FUNCTION_BLOCK FB_XtsXlMoverUtility
VAR_INPUT
	EdtDriverOid: OTCID;
END_VAR

VAR_OUTPUT
	bBusy: BOOL;
	bDone: BOOL;
	bError: BOOL;
	bInit: BOOL;
	ipResultMessage: I_TcMessage := fbResult;
END_VAR

VAR
	fbResult: FB_TcMessage;
	_ipComObject: ITComObject;
	
	PID_TriggerLeave						: PTCID := 16#030802EF;
	PID_TriggerArrive						: PTCID := 16#030802EE;
	PID_IsVirtualFeedbackEnabled			: PTCID := 16#0308050B;
	PID_ConfiguredDetectionTrackObjectId	: PTCID := 16#030802F0;
	PID_StartupTrackPosition				: PTCID := 16#03080370;
END_VAR

IF NOT bInit THEN
	IF GetComObject(nObjectId:=EdtDriverOid) THEN
		bInit:=TRUE;
	END_IF
	RETURN;
END_IF

METHOD GetComObject : BOOL
VAR_INPUT
	nObjectId: OTCID;
END_VAR
IF FW_ObjMgr_GetObjectInstance(	oid		:= nObjectId, 
								iid		:= TC_GLOBAL_IID_LIST.IID_ITComObject, 
								pipUnk	:= ADR(_ipComObject)) = 0
THEN
	GetComObject := TRUE;
END_IF
END_METHOD

METHOD SetConfiguredDetectionTrackObjectId : BOOL
VAR_INPUT
	nConfiguredDetectionTrackObjectId: OTCID;
END_VAR

VAR
	nValue: OTCID;
	stEventEntry: TcEventEntry;
	pstEventEntry: REFERENCE TO TcEventEntry := stEventEntry;
END_VAR

VAR_INST
	hResult : HRESULT;
END_VAR
bError := FALSE;

nValue := nConfiguredDetectionTrackObjectId;

IF _ipComObject <> 0 THEN 
	 hResult := 	_ipComObject.TcSetObjPara(		pid := PID_ConfiguredDetectionTrackObjectId,
													nData := SIZEOF(nValue),
													pData := ADR(nValue),
													pgp := 0); 	
	IF hResult = 0 THEN
		SetConfiguredDetectionTrackObjectId := TRUE;
	ELSE
		HRESULTAdsErr_TO_TcEventEntry(hResult,stEventEntry);
		IF NOT fbResult.EqualsToEventEntryEx( stOther := stEventEntry) THEN
			fbResult.CreateEx(stEventEntry, 0);
			fbResult.Send(0);
			fbResult.Release();
		END_IF
		bError := TRUE;
	END_IF							
END_IF
END_METHOD

METHOD SetIsVirtualFeedbackEnabled : BOOL
VAR_INPUT
	bSetIsVirtualFeedbackEnabled: BOOL;
END_VAR

VAR
	nValue: BOOL;
	stEventEntry: TcEventEntry;
	pstEventEntry: REFERENCE TO TcEventEntry := stEventEntry;
END_VAR

VAR_INST
	hResult : HRESULT;
END_VAR
bError := FALSE;

nValue := bSetIsVirtualFeedbackEnabled;

IF _ipComObject <> 0 THEN 
	 hResult := 	_ipComObject.TcSetObjPara(		pid := PID_IsVirtualFeedbackEnabled,
													nData := SIZEOF(nValue),
													pData := ADR(nValue),
													pgp := 0); 	
	IF hResult = 0 THEN
		SetIsVirtualFeedbackEnabled := TRUE;
	ELSE
		HRESULTAdsErr_TO_TcEventEntry(hResult,stEventEntry);
		IF NOT fbResult.EqualsToEventEntryEx( stOther := stEventEntry) THEN
			fbResult.CreateEx(stEventEntry, 0);
			fbResult.Send(0);
			fbResult.Release();
		END_IF
		bError := TRUE;
	END_IF							
END_IF
END_METHOD

METHOD SetStartupTrackPosition : BOOL
VAR_INPUT
	nStartupTrackPosition: REAL;
END_VAR

VAR
	nValue: REAL;
	stEventEntry: TcEventEntry;
	pstEventEntry: REFERENCE TO TcEventEntry := stEventEntry;
END_VAR

VAR_INST
	hResult : HRESULT;
END_VAR
bError := FALSE;

nValue := nStartupTrackPosition;

IF _ipComObject <> 0 THEN 
	 hResult := 	_ipComObject.TcSetObjPara(		pid := PID_StartupTrackPosition,
													nData := SIZEOF(nValue),
													pData := ADR(nValue),
													pgp := 0); 	
	IF hResult = 0 THEN
		SetStartupTrackPosition := TRUE;
	ELSE
		HRESULTAdsErr_TO_TcEventEntry(hResult,stEventEntry);
		IF NOT fbResult.EqualsToEventEntryEx( stOther := stEventEntry) THEN
			fbResult.CreateEx(stEventEntry, 0);
			fbResult.Send(0);
			fbResult.Release();
		END_IF
		bError := TRUE;
	END_IF							
END_IF
END_METHOD

METHOD TriggerArrive : BOOL
VAR_INPUT
END_VAR

VAR
	nValue: BOOL;
	stEventEntry: TcEventEntry;
	pstEventEntry: REFERENCE TO TcEventEntry := stEventEntry;
END_VAR

VAR_INST
	hResult : HRESULT;
END_VAR
//bError := FALSE;

nValue := TRUE;

IF _ipComObject <> 0 THEN 
	 hResult := 	_ipComObject.TcSetObjPara(		pid := PID_TriggerArrive,
													nData := SIZEOF(nValue),
													pData := ADR(nValue),
													pgp := 0); 	
	IF hResult = 0 THEN
		TriggerArrive := TRUE;
	ELSE
		HRESULTAdsErr_TO_TcEventEntry(hResult,stEventEntry);
		IF NOT fbResult.EqualsToEventEntryEx( stOther := stEventEntry) THEN
			fbResult.CreateEx(stEventEntry, 0);
			fbResult.Send(0);
			fbResult.Release();
		END_IF
		bError := TRUE;
		TriggerArrive := FALSE;
	END_IF							
END_IF
END_METHOD

METHOD TriggerLeave : BOOL
VAR_INPUT
END_VAR

VAR
	nValue: BOOL;
	stEventEntry: TcEventEntry;
	pstEventEntry: REFERENCE TO TcEventEntry := stEventEntry;
END_VAR

VAR_INST
	hResult : HRESULT;
END_VAR
bError := FALSE;

nValue := TRUE;

IF _ipComObject <> 0 THEN 
	 hResult := 	_ipComObject.TcSetObjPara(		pid := PID_TriggerLeave,
													nData := SIZEOF(nValue),
													pData := ADR(nValue),
													pgp := 0); 	
	IF hResult = 0 THEN
		TriggerLeave := TRUE;
	ELSE
		HRESULTAdsErr_TO_TcEventEntry(hResult,stEventEntry);
		IF NOT fbResult.EqualsToEventEntryEx( stOther := stEventEntry) THEN
			fbResult.CreateEx(stEventEntry, 0);
			fbResult.Send(0);
			fbResult.Release();
		END_IF
		bError := TRUE;
	END_IF							
END_IF
END_METHOD

END_FUNCTION_BLOCK

(* stored: Version 1.1.0.1, ProductVersion 3.1.4026.8
   POU FB_XtsXlMoverUtility: Id {187f933d-eac3-44fd-a785-99f141def362}, SpecialFunc None
   Method GetComObject: Id {3bab5b9c-2b0e-451c-bdae-5b68d9d01859}
   Method SetConfiguredDetectionTrackObjectId: Id {01ced642-e3b1-4ad2-a438-0d6fa4c980df}
   Method SetIsVirtualFeedbackEnabled: Id {107284cf-c52b-42fc-bf5a-5dfba57bccf7}
   Method SetStartupTrackPosition: Id {79d30cc9-e7ba-49d7-9966-b740df7c960b}
   Method TriggerArrive: Id {ff515d71-ba62-4ca9-a248-bf49d1d44595}
   Method TriggerLeave: Id {ad6fe72b-e1fc-4783-9f84-81d8f4fda188} *)
